// TIA Portal V20 export
TYPE "LBP_typeMcp310PnOutput"
TITLE = MCP 310 PN image / Image du MCP 310 PN
// Output image of MCP 310 PN / Image de sortie du MCP 310 PN
   STRUCT
      standard { S7_SetPoint := 'True'} : "LBP_typeMcp310StandardOutput";   // Output image of MCP 310 / Image de sortie du MCP 310
   END_STRUCT;
END_TYPE
